Staubli VAL3: MX1_COMMANDS.pjx

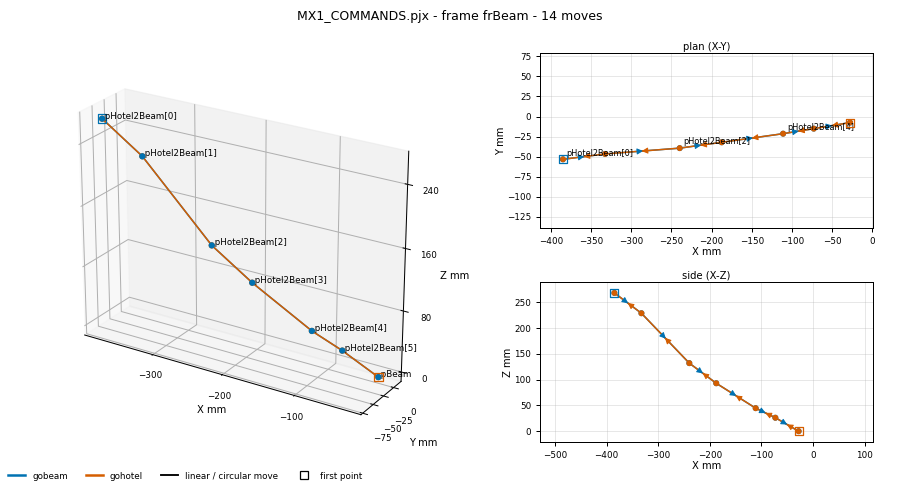
[picture p0: tool path of MX1_COMMANDS.pjx in frame frBeam, 14 of 32 moves have a stored position in this frame; points joined in program order, loops and branches not executed]
--- MX1_COMMANDS.pjx ---
Parameters version=s7.9.4 stackSize=5000 millimeterUnit=true
Program file=changeToolMove.pgx
Program file=deleteMove.pgx
Program file=external.pgx
Program file=getX.pgx
Program file=getY.pgx
Program file=getZ.pgx
Program file=goBeam.pgx
Program file=goHotel.pgx
Program file=gripper.pgx
Program file=isSettled.pgx
Program file=moveX.pgx
Program file=moveY.pgx
Program file=moveZ.pgx
Program file=pickPlate.pgx
Program file=placePlate.pgx
Program file=power.pgx
Program file=restartMove.pgx
Program file=setFrame.pgx
Program file=setTool.pgx
Program file=setup.pgx
Program file=start.pgx
Program file=stop.pgx
Program file=stopMove.pgx
Data file=MX1_COMMANDS.dtx
Library alias=io path=Disk://io autoload=true password=
Library alias=external path=Disk://external autoload=true password=

--- MX1_COMMANDS.dtx ---
frame frActive = {fatherId=world[0]}
frame frBeam = {x=-161.188459, y=496.371638, z=-199.667625, rx=3.214523, ry=3.0212331, rz=133.562606, fatherId=world[0]}
frame frHotel = {x=286.392398, y=319.87105, z=42.0189883, rx=90.184146, ry=-45.0765197, rz=-89.806008, fatherId=world[0]}
frame frRack = {x=-153.788748, y=277.287549, z=-206.151597, rx=-0.378549, ry=-0.11222, rz=142.369658, fatherId=world[0]}
jointRx jHome = {j1=-150.761388, j2=-6.734913, j3=85.0824661, j4=133.894848, j5=36.278934, j6=59.830326}
mdesc mNomSpeed = {blend=off}
num nHoldingPlate
pointRx pBeam = {x=-27.723888, y=-7.540843, z=-0.00401315, rx=78.213789, ry=94.16282, rz=9.733183, fatherId=frBeam[0]}
pointRx pDest = {x=418.887279, y=-94.568514, z=-308.425583, rx=89.522984, ry=76.446497, rz=-90.78804, shoulder=lefty, elbow=epositive, wrist=wnegative, fatherId=frActive[0]}
pointRx pHotel[11]
  [0] = {x=-125.524742, y=32.928965, z=129.506951, rx=-1.0716474, ry=-179.57369, rz=-2.748198, fatherId=frHotel[0]}
  [1] = {x=-9.734034, y=32.928818, z=-9.820607, rx=-1.0710121, ry=-179.574275, rz=-2.749031, fatherId=frHotel[0]}
  [2] = {x=20.265022, y=32.928818, z=-9.820607, rx=-1.0709964, ry=-179.575149, rz=-2.74904, fatherId=frHotel[0]}
  [3] = {x=50.265702, y=32.928818, z=-9.820607, rx=-1.0709978, ry=-179.575302, rz=-2.74904, fatherId=frHotel[0]}
  [4] = {x=80.27455, y=32.928818, z=-9.820607, rx=-1.071003, ry=-179.576432, rz=-2.749042, fatherId=frHotel[0]}
  [5] = {x=110.270191, y=29.547911, z=-9.820606, rx=-0.13897, ry=-179.575262, rz=-2.748802, fatherId=frHotel[0]}
  [6] = {x=140.267371, y=29.547911, z=-9.820606, rx=-0.138766, ry=-179.576262, rz=-2.748899, fatherId=frHotel[0]}
  [7] = {x=170.267085, y=29.547911, z=-9.820606, rx=-0.138781, ry=-179.577185, rz=-2.748913, fatherId=frHotel[0]}
  [8] = {x=200.273264, y=29.547911, z=-9.820607, rx=-0.138807, ry=-179.577334, rz=-2.748906, fatherId=frHotel[0]}
  [9] = {x=230.274778, y=29.547911, z=-9.820607, rx=-0.138782, ry=-179.57707, rz=-2.748908, fatherId=frHotel[0]}
  [10] = {x=260.273406, y=29.547911, z=-9.820608, rx=-0.138774, ry=-179.577066, rz=-2.748909, fatherId=frHotel[0]}
pointRx pHotel2Beam[6]
  [0] = {x=-384.885169, y=-53.248704, z=267.993956, rx=90.449128, ry=21.634862, rz=84.812396, fatherId=frBeam[0]}
  [1] = {x=-332.447311, y=-46.537661, z=228.647356, rx=90.832753, ry=30.739376, rz=82.63404, fatherId=frBeam[0]}
  [2] = {x=-239.633325, y=-39.352015, z=131.894801, rx=96.322781, ry=51.214932, rz=79.135034, fatherId=frBeam[0]}
  [3] = {x=-187.422675, y=-32.0850414, z=92.941008, rx=102.48851, ry=61.97177, rz=75.962643, fatherId=frBeam[0]}
  [4] = {x=-110.99078, y=-21.362599, z=44.619423, rx=111.0248449, ry=76.977395, rz=-21.203897, fatherId=frBeam[0]}
  [5] = {x=-72.833062, y=-15.0880081, z=26.115733, rx=76.58185, ry=93.958531, rz=12.261834, fatherId=frBeam[0]}
pointRx pOBeam = {x=-161.18892, y=496.371418, z=-199.66767, rx=-89.164201, ry=-50.51892, rz=179.308757, fatherId=world[0]}
pointRx pOHotel = {x=286.150494, y=319.693132, z=42.0716019, rx=-88.412511, ry=44.721115, rz=-159.366909, fatherId=world[0]}
pointRx pORack = {x=-153.788748, y=277.287549, z=-206.151597, rx=-178.912895, ry=-0.558319, rz=51.4705, fatherId=world[0]}
pointRx pRack[5]
  [0] = {x=0.00130708, y=124.49452, z=181.38133, rx=-0.806017, ry=178.698036, rz=15.344641, fatherId=frRack[0]}
  [1] = {fatherId=frRack[0]}
  [2] = {fatherId=frRack[0]}
  [3] = {fatherId=frRack[0]}
  [4] = {fatherId=frRack[0]}
pointRx pXBeam = {x=-224.31737, y=562.552126, z=-192.611505, rx=88.595611, ry=-131.0118701, rz=-3.207831, fatherId=world[0]}
pointRx pXHotel = {x=287.0377751, y=320.0914829, z=-227.908852, rx=-88.413524, ry=44.720978, rz=-159.365948, fatherId=world[0]}
pointRx pXRack = {x=-284.997921, y=378.43924, z=-207.0769021, rx=-178.913758, ry=-0.557885, rz=51.470771, fatherId=world[0]}
pointRx pYBeam = {x=-337.991927, y=449.17776, z=-192.974679, rx=88.594452, ry=-131.011574, rz=-3.208841, fatherId=world[0]}
pointRx pYHotel = {x=328.883072, y=278.133406, z=-227.708715, rx=-88.413466, ry=44.721523, rz=-159.366478, fatherId=world[0]}
pointRx pYRack = {x=-403.395202, y=216.566045, z=-206.2393, rx=-178.913669, ry=-0.557283, rz=51.471015, fatherId=world[0]}
sio sTest = {link=Socket\sock1}
tool tActive = {fatherId=flange[0], ioLink=valve1}
tool tGripper = {fatherId=flange[0], ioLink=valve1}
trsf trPickPlateHor = {x=6, z=-145}
trsf trPickPlateVer = {x=6}

--- start.pgx ---
program start()
  local num i
  local num nBuffer[1 30]
  local num nbc[30 1]
  local num ndf[30 1 1]
  local num nt[30]
  local string sBufer
begin
  //call external:start()
  //pDest=here(tActive,frActive)
end

--- changeToolMove.pgx ---
public program changeToolMove(num nChange (dimensions=1))
begin
  call external:oGripCmd2(nChange)
end

--- deleteMove.pgx ---
public program deleteMove()
begin
  resetMotion()
  pDest=here(tActive,frActive)
end

--- external.pgx ---
public program external()
begin
  call external:start()
end

--- getX.pgx ---
public program getX(num& nValueX (dimensions=1))
  local point pHere
begin
  pHere=here(tActive,frActive)
  nValueX=pHere.trsf.x
end

--- getY.pgx ---
public program getY(num& nValueY (dimensions=1))
  local point pHere
begin
  pHere=here(tActive,frActive)
  nValueY=pHere.trsf.y
end

--- getZ.pgx ---
public program getZ(num& nValueZ (dimensions=1))
  local point pHere
begin
  pHere=here(tActive,frActive)
  nValueZ=pHere.trsf.z
end

--- goBeam.pgx ---
program goBeam()
begin
  //FUTURE ADJUSTMENT: argument nFrom
  //nFrom = 0 -> Dewar to Beam
  //nFrom = 1 -> Hotel to Beam
  movel(pHotel[0],flange,mNomSpeed)
  movel(pHotel2Beam[0],flange,mNomSpeed)
  movel(pHotel2Beam[1],flange,mNomSpeed)
  movel(pHotel2Beam[2],flange,mNomSpeed)
  movel(pHotel2Beam[3],flange,mNomSpeed)
  movel(pHotel2Beam[4],flange,mNomSpeed)
  movel(pHotel2Beam[5],flange,mNomSpeed)
  movel(pBeam,flange,mNomSpeed)
end

--- goHotel.pgx ---
program goHotel(num nFrom (dimensions=1))
  local trsf movHorizontal
begin
  //FUTURE ADJUSTMENT: argument nFrom
  //nFrom = 0 -> jHome or pHotel [0] to pHotel[0]
  //nFrom = 1 -> pBeam to pHotel[0]
  switch nFrom
    case 0
      movel(pHotel[0],flange,mNomSpeed)
    break
    case 1
      movel(pBeam,flange,mNomSpeed)
      movel(pHotel2Beam[5],flange,mNomSpeed)
      movel(pHotel2Beam[4],flange,mNomSpeed)
      movel(pHotel2Beam[3],flange,mNomSpeed)
      movel(pHotel2Beam[2],flange,mNomSpeed)
      movel(pHotel2Beam[1],flange,mNomSpeed)
      movel(pHotel2Beam[0],flange,mNomSpeed)
      movel(pHotel[0],flange,mNomSpeed)
    break
    default
      popUpMsg("error goHotel: nFrom"+chr(nFrom))
    break
  endSwitch
  waitEndMove()
end

--- gripper.pgx ---
public program gripper(num nOpen (dimensions=1))
begin
  //nOpen = 0 - close gripper
  //nOpen = 1 - open gripper
  //
  switch nOpen
    case 0
      close(flange)
    break
    case 1
      open(flange)
    break
    default
      logMsg("gripper(): nOpen = "+toString("",nOpen))
    break
  endSwitch
end

--- isSettled.pgx ---
public program isSettled(num& nSettled (dimensions=1))
  local bool bSettled
begin
  //robot moving = return 1/isSettled = false
  //robot stopped = return 0/isSettled = false
  bSettled=isSettled()
  switch bSettled
    case true
      nSettled=0
    break
    case false
      nSettled=1
    break
    default
      logMsg("error isSettled")
    break
  endSwitch
end

--- moveX.pgx ---
public program moveX(num nDx (dimensions=1))
  local point pFinal
  local point pHere
begin
  //pHere=here(tActive,frActive)
  //pFinal=compose(pHere,frActive,{nDx,0,0,0,0,0})
  pDest=compose(pDest,frActive,{nDx,0,0,0,0,0})
  //movel(pFinal,tActive,mNomSpeed)
  movel(pDest,tActive,mNomSpeed)
end

--- moveY.pgx ---
public program moveY(num nDy (dimensions=1))
  local point pFinal
  local point pHere
begin
  //pHere=here(tActive,frActive)
  //pFinal=compose(pHere,frActive,{0,nDy,0,0,0,0})
  //movel(pFinal,tActive,mNomSpeed)
  pDest=compose(pDest,frActive,{0,nDy,0,0,0,0})
  movel(pDest,tActive,mNomSpeed)
end

--- moveZ.pgx ---
public program moveZ(num nDz (dimensions=1))
  local frame frActual
  local point pFinal
  local point pHere
begin
  pHere=here(tActive,frActive)
  pFinal=compose(pHere,frActive,{0,0,nDz,0,0,0})
  movel(pFinal,tActive,mNomSpeed)
end

--- pickPlate.pgx ---
public program pickPlate(num nPlate (dimensions=1))
begin
  //robot at pHotel[0] or jHome
  call goHotel(0)
  open(flange)
  movel(appro(pHotel[nPlate],trPickPlateHor),flange,mNomSpeed)
  movel(appro(pHotel[nPlate],trPickPlateVer),flange,mNomSpeed)
  movel(pHotel[nPlate],flange,mNomSpeed)
  close(flange)
  delay(1)
  movel(appro(pHotel[nPlate],trPickPlateVer),flange,mNomSpeed)
  movel(appro(pHotel[nPlate],trPickPlateHor),flange,mNomSpeed)
  movel(pHotel[0],flange,mNomSpeed)
  waitEndMove()
  nHoldingPlate=nPlate
end

--- placePlate.pgx ---
public program placePlate(num nPlate (dimensions=1))
begin
  //ADJUSTMENT: chance goHotel argument
  //when test phase is over (0 to 1)
  //robot supposed to be at Beam (goHotel(1))
  call goHotel(1)
  movel(appro(pHotel[nHoldingPlate],trPickPlateHor),flange,mNomSpeed)
  movel(appro(pHotel[nHoldingPlate],trPickPlateVer),flange,mNomSpeed)
  movel(pHotel[nHoldingPlate],flange,mNomSpeed)
  open(flange)
  delay(1)
  movel(appro(pHotel[nHoldingPlate],trPickPlateVer),flange,mNomSpeed)
  movel(appro(pHotel[nHoldingPlate],trPickPlateHor),flange,mNomSpeed)
  movel(pHotel[0],flange,mNomSpeed)
  waitEndMove()
  nHoldingPlate=0
end

--- power.pgx ---
public program power(num nPower (dimensions=1))
begin
  //0  to disable power
  //1  to enable power
  switch nPower
    case 0
      disablePower()
    break
    case 1
      enablePower()
    break
    default
      logMsg("power: argumento invalido"+chr(nPower))
    break
  endSwitch
end

--- restartMove.pgx ---
public program restartMove()
begin
  restartMove()
end

--- setFrame.pgx ---
public program setFrame(num nFrame (dimensions=1))
begin
  switch nFrame
    case 0
      frActive=world
    break
    case 1
      frActive=frHotel
    break
    case 2
      frActive=frBeam
    break
    case 3
      frActive=frRack
    break
    default
      logMsg("erro setFrame: "+chr(nFrame))
    break
  endSwitch
end

--- setTool.pgx ---
public program setTool(num nTool (dimensions=1))
begin
  switch nTool
    case 0
      tActive=flange
    break
    case 1
      tActive=tGripper
    break
    case 2
    break
    default
      logMsg("erro setTool: "+chr(nTool))
    break
  endSwitch
end

--- stopMove.pgx ---
public program stopMove()
begin
  stopMove()
end
